// TIA Portal V18 export
FUNCTION_BLOCK "ST10_Flow14_B2Press"   // FB1084, GRAPH
// stored: AcknowledgeErrorsRequired false, AutoNumber false, GraphVersion 6.0, InitialValuesAcquisition false, SetENOAutomatically false
   // inherited from GRAPH_BASE
   VAR_INPUT
      iSysInface : "RCS_SysComInterface_V1";
   END_VAR
   VAR_IN_OUT
      ioPM_Inface : "RCS_PMInterface_V1";
      ioStatus : Int;
   END_VAR
   VAR
      sCtrlMode { S7_SetPoint := 'True'} : "SysFlowCtrlGraph";
      sUpdMES_Data : Bool;   // 更新MES数据
      工件放行中 : Bool;
      前站站号 { ExternalAccessible := 'False'; ExternalVisible := 'False'; ExternalWritable := 'False'} : UInt;
      本站站号 { ExternalAccessible := 'False'; ExternalVisible := 'False'; ExternalWritable := 'False'} : UInt;
      弹窗Temp : Array[1..10] of Int;
      AlarmID : Int;
      TON { S7_SetPoint := 'True'} : Array[0..10] of TON_TIME;
      TOF { S7_SetPoint := 'True'} : Array[0..10] of TOF_TIME;
      sUP { S7_SetPoint := 'True'} : Array[0..10] of Bool;
      更新RFID完成 : Bool;
   END_VAR
   VAR_TEMP
      Tempresult : USInt;
      本站站号乘10 : UInt;
   END_VAR
   // // TON[0] : 托盘流入1托盘到位传感器 / iA-Rotating product Check
   // // TON[1] : 托盘流入1托盘到位传感器
   // // TON[2] : 托盘流入1产品有无传感器
   // // TON[3] : 托盘流入1产品有无传感器
   // // TON[4] : 托盘流入1姿态检测光电2
   // // TON[5] : 托盘流入1姿态检测光电3
   // // TON[0].Q : 托盘流入1托盘到位 / iA-Rotating product Check
   // // TON[1].Q : 托盘流入1托盘无
   // // TON[2].Q : 托盘流入1有产品
   // // TON[3].Q : 托盘流入1无产品
   // // TON[4].Q : 托盘流入1姿态检测光电2
   // // TON[5].Q : 托盘流入1姿态检测光电3
   // // TOF[1] : iA-Rotating product Check
BEGIN
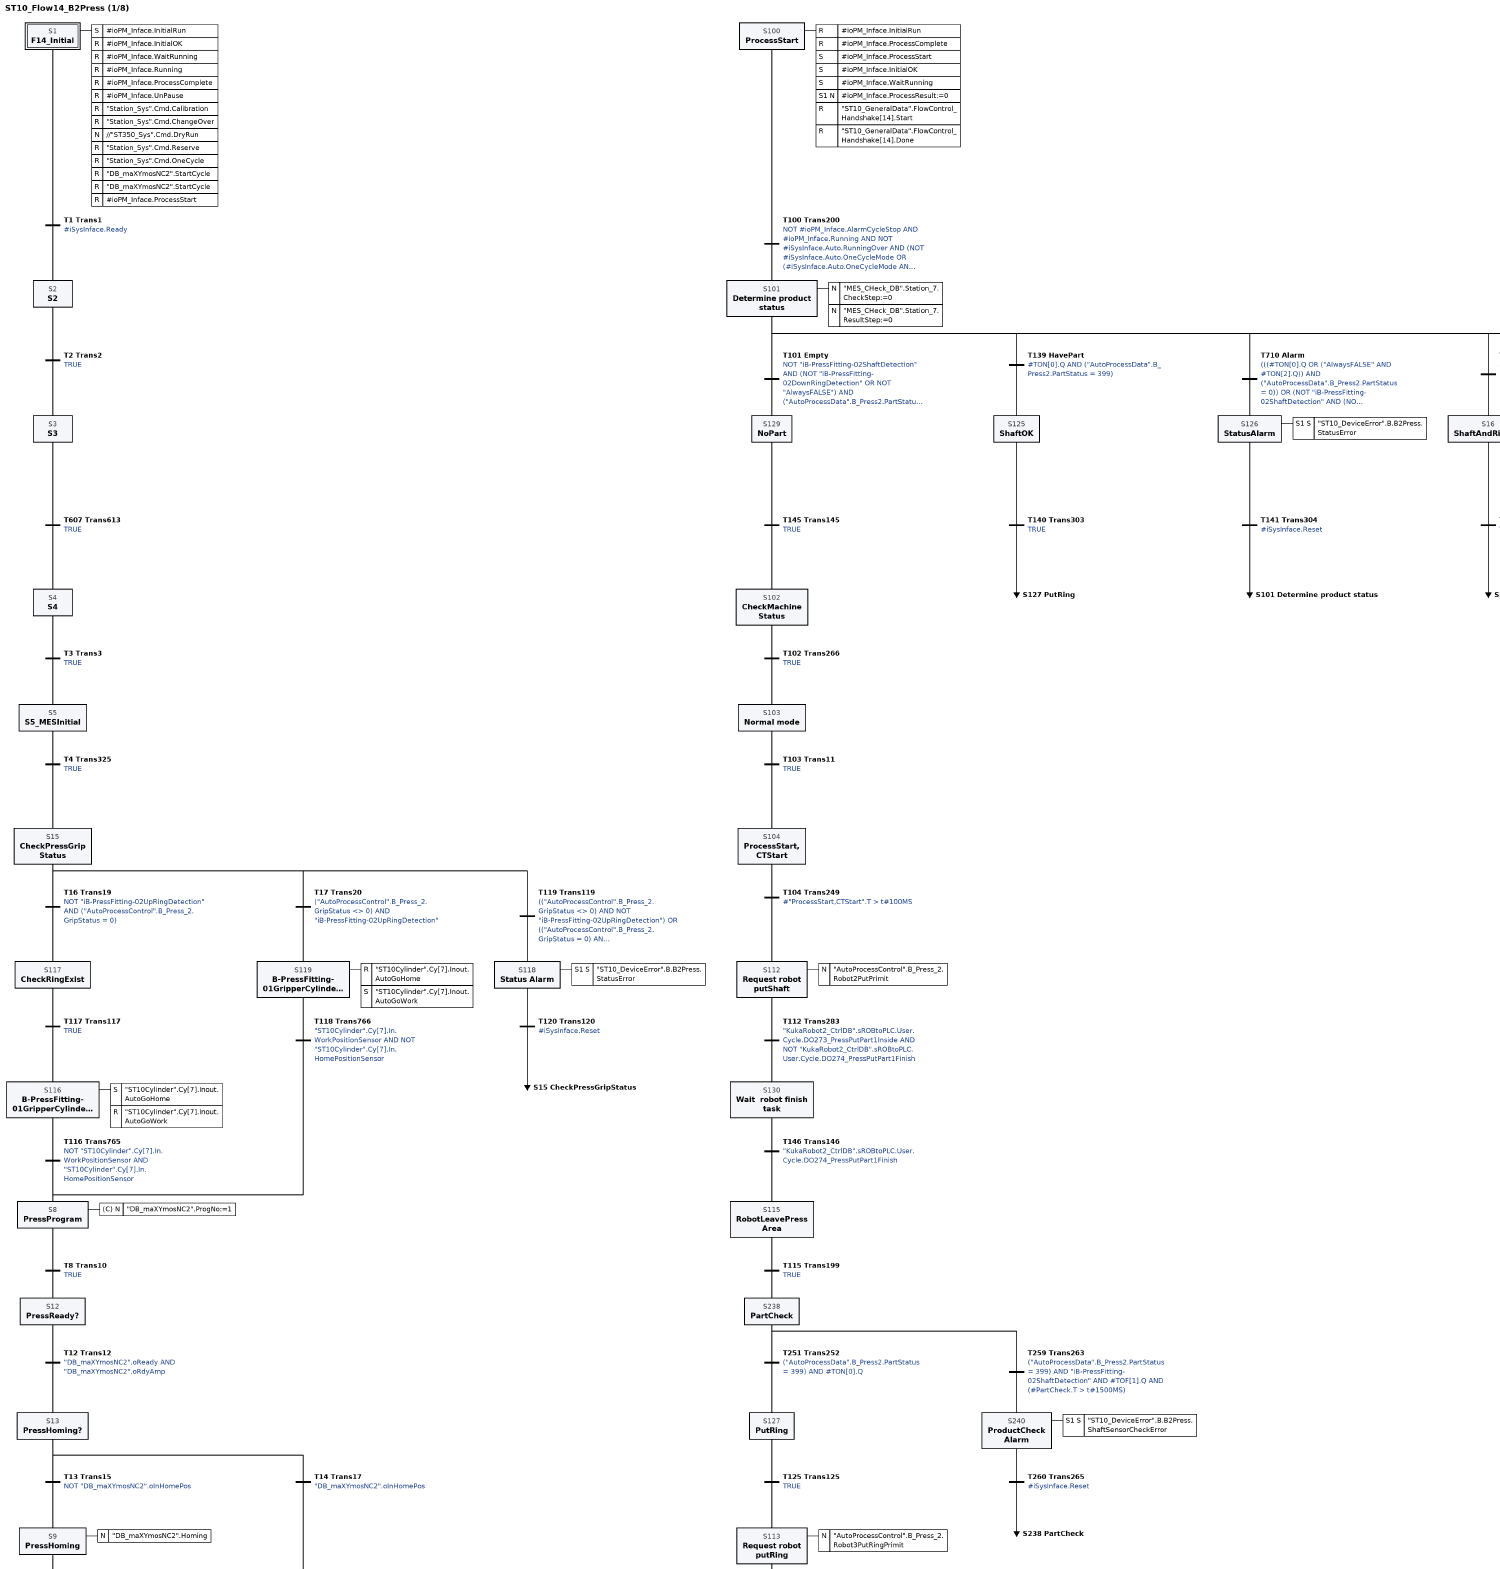
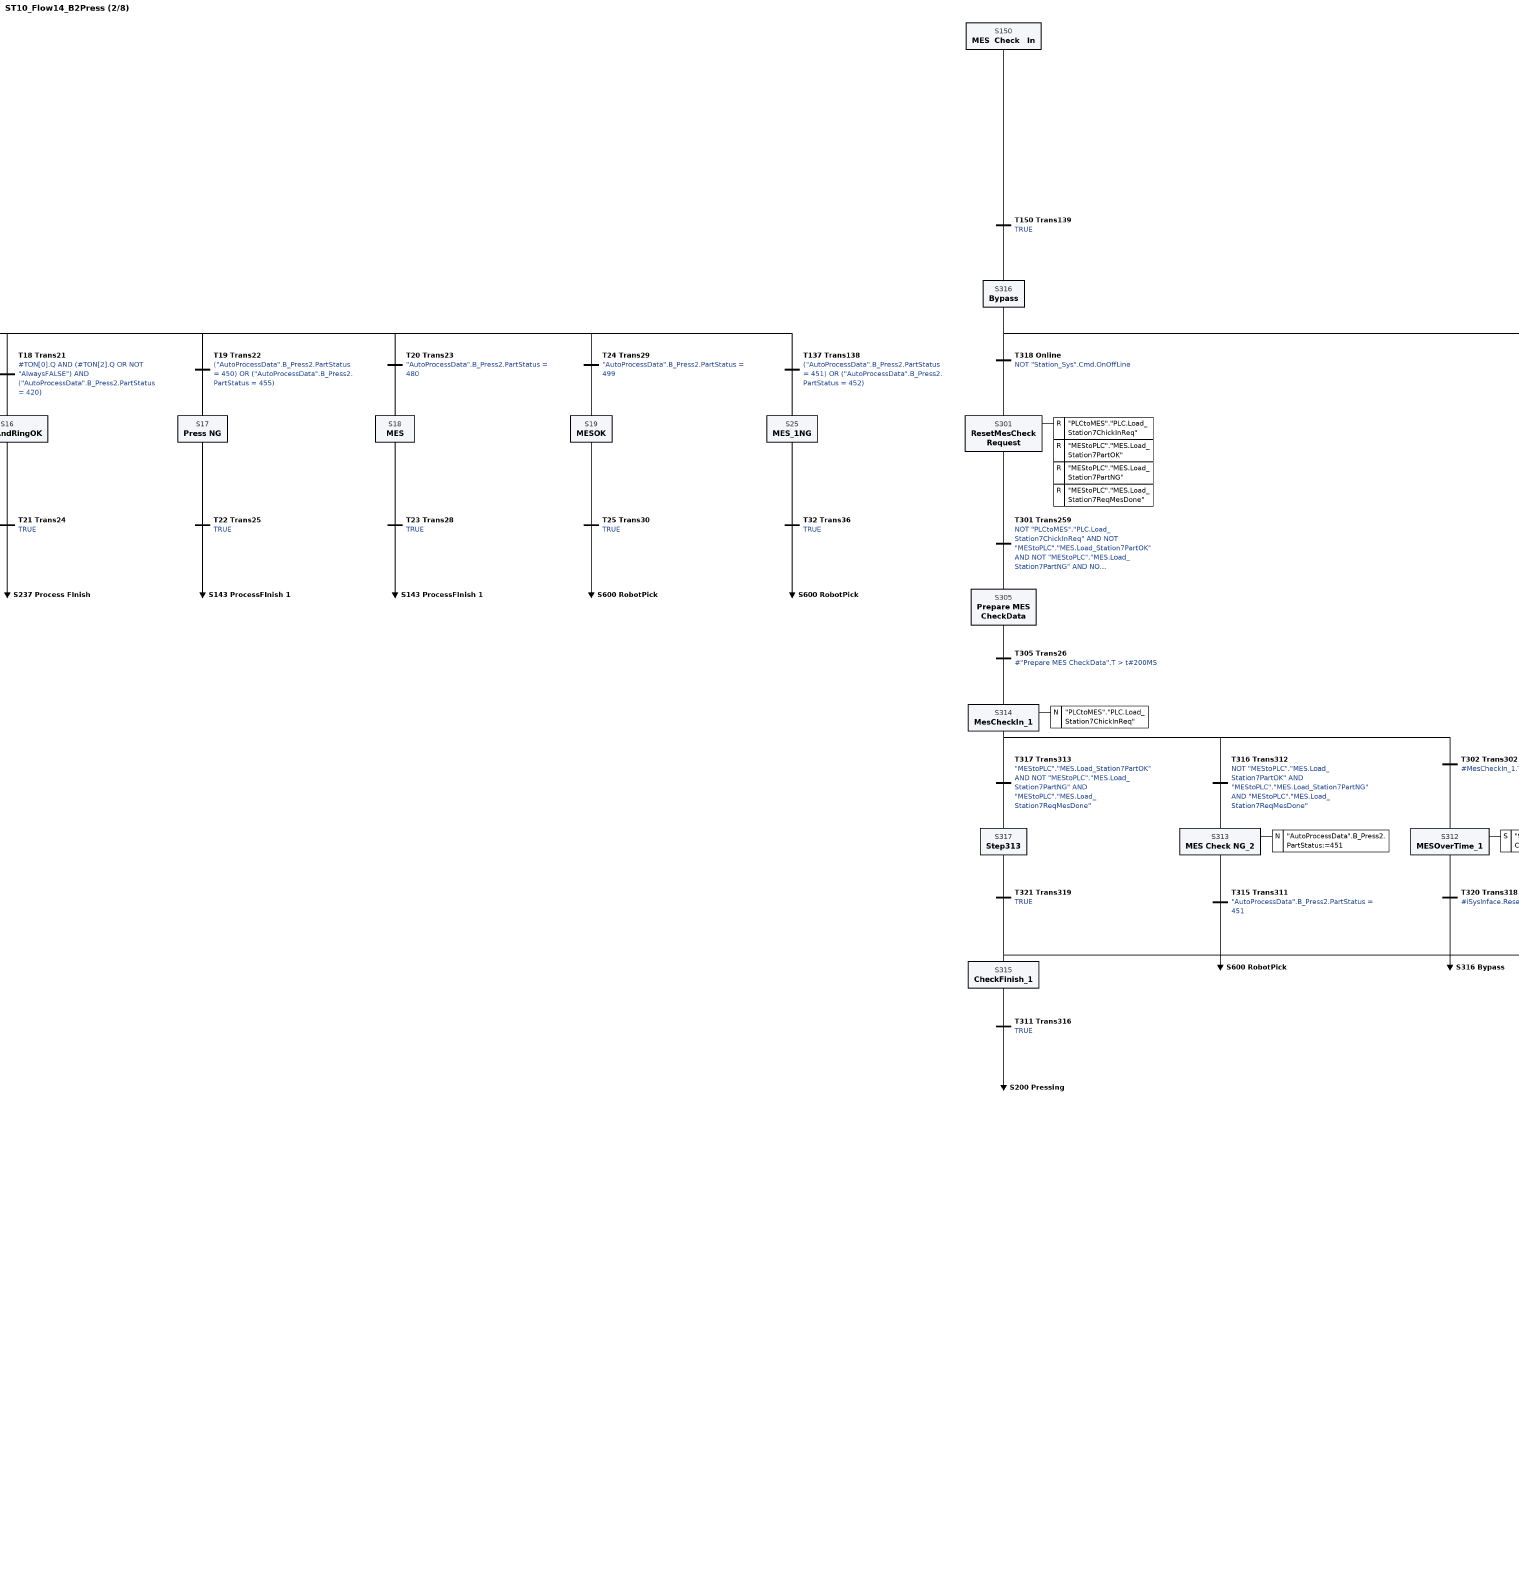
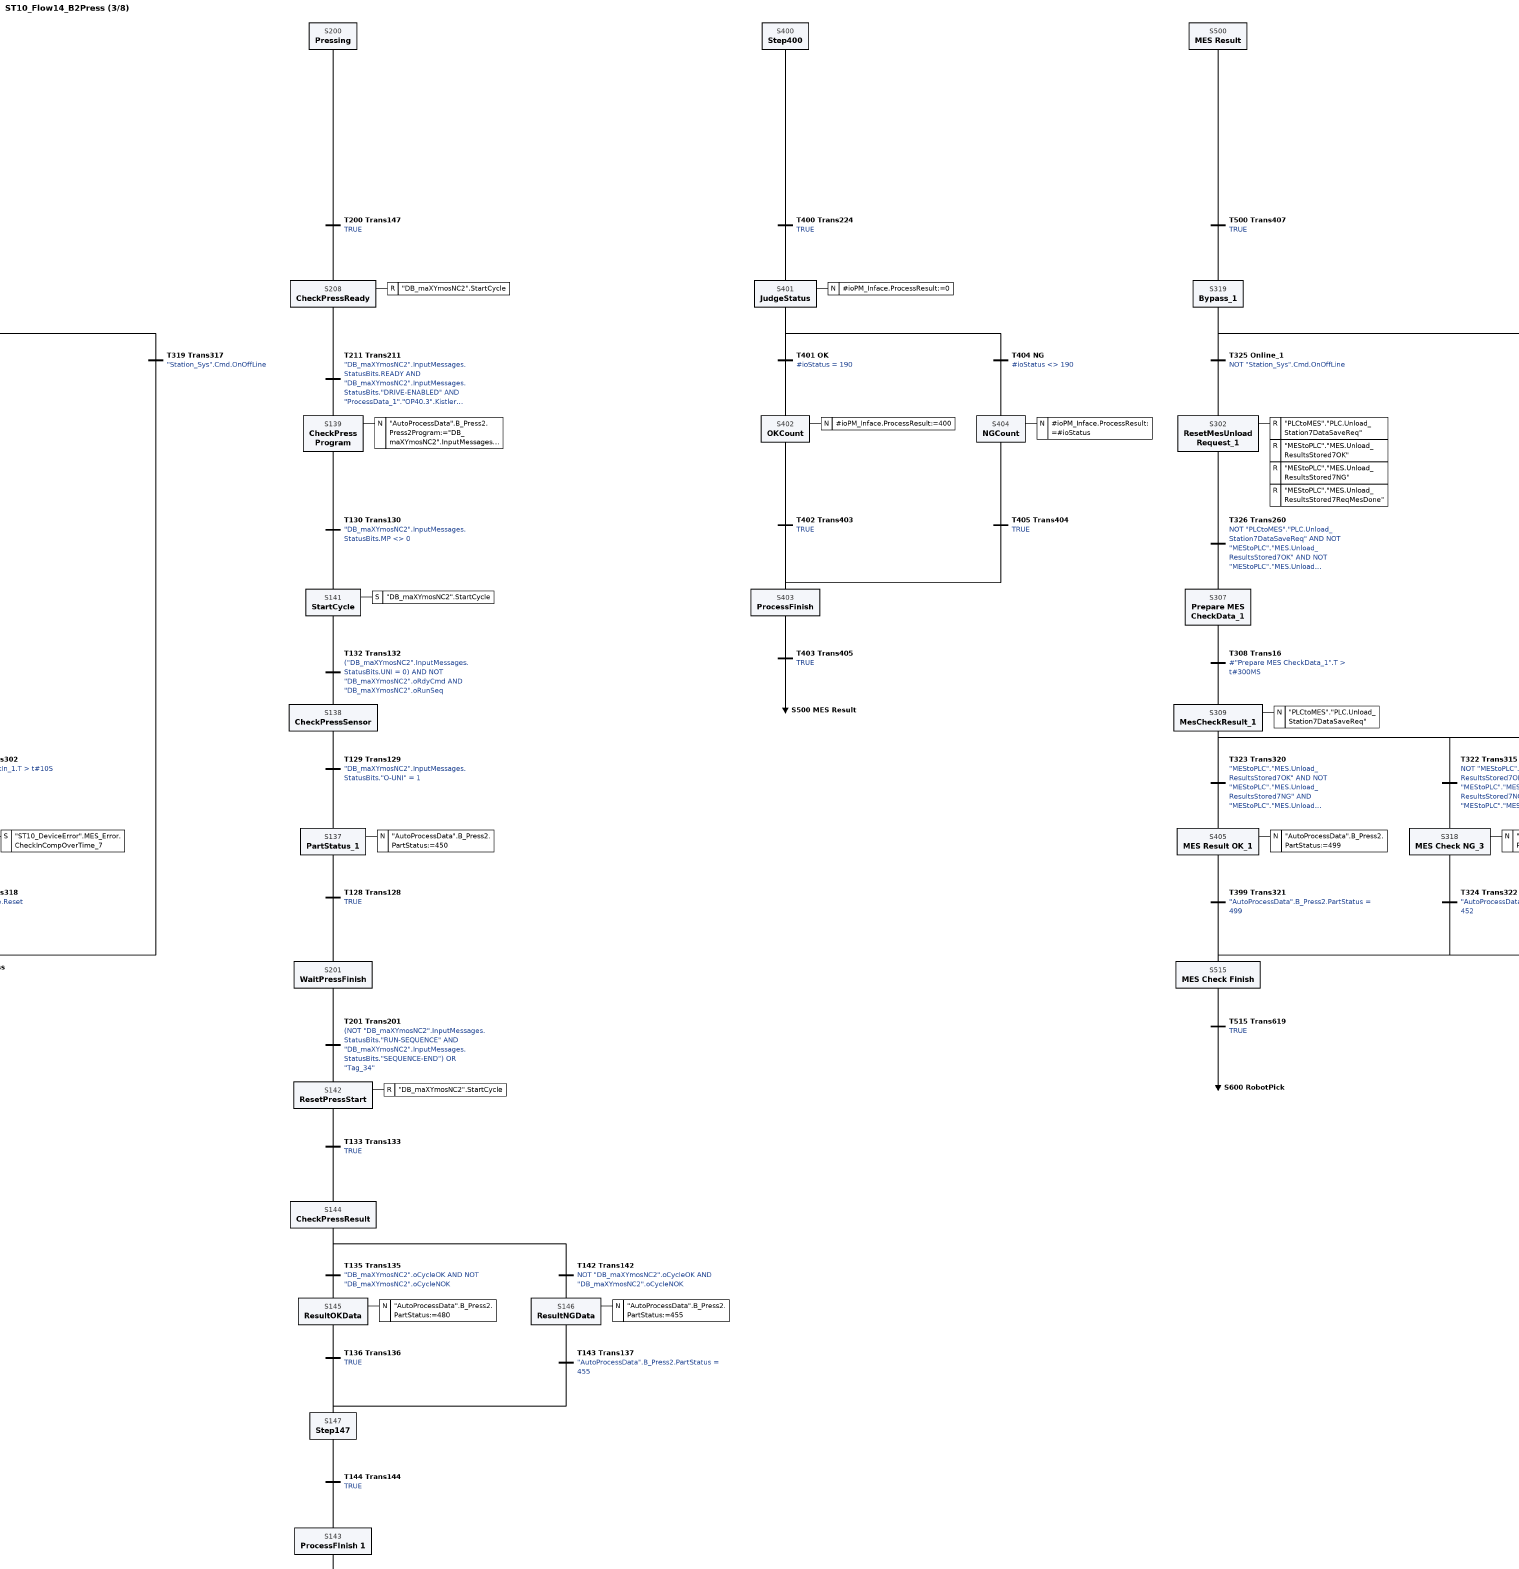
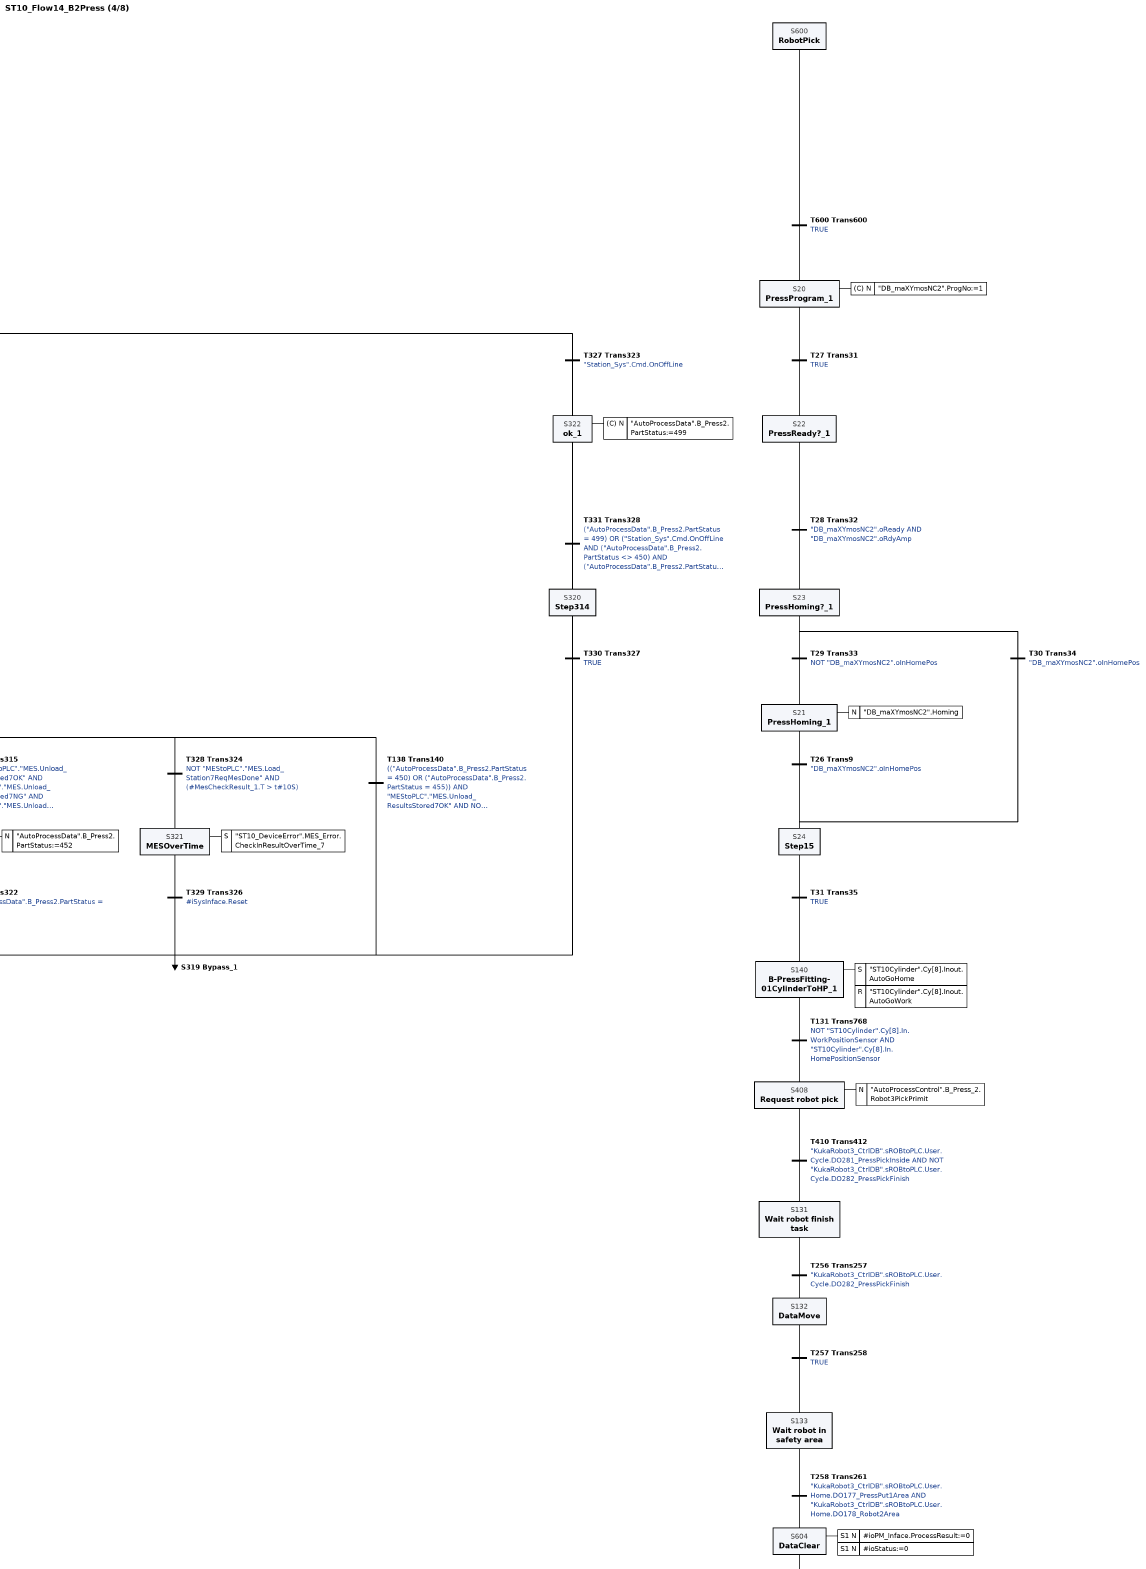
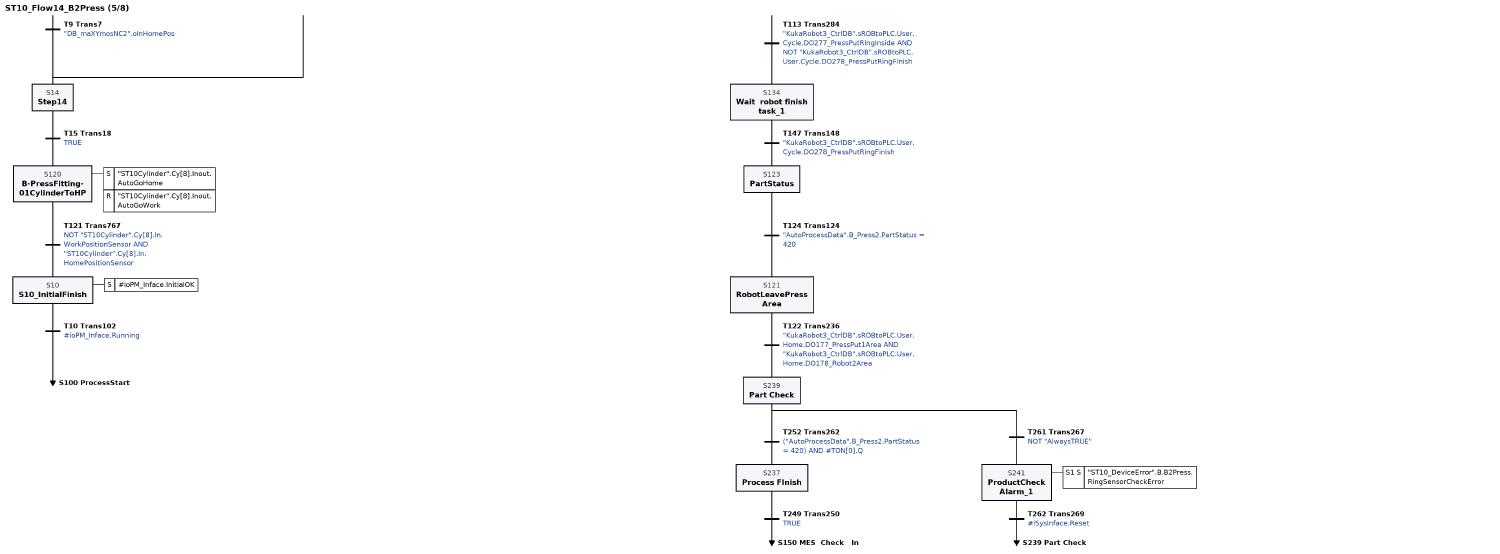
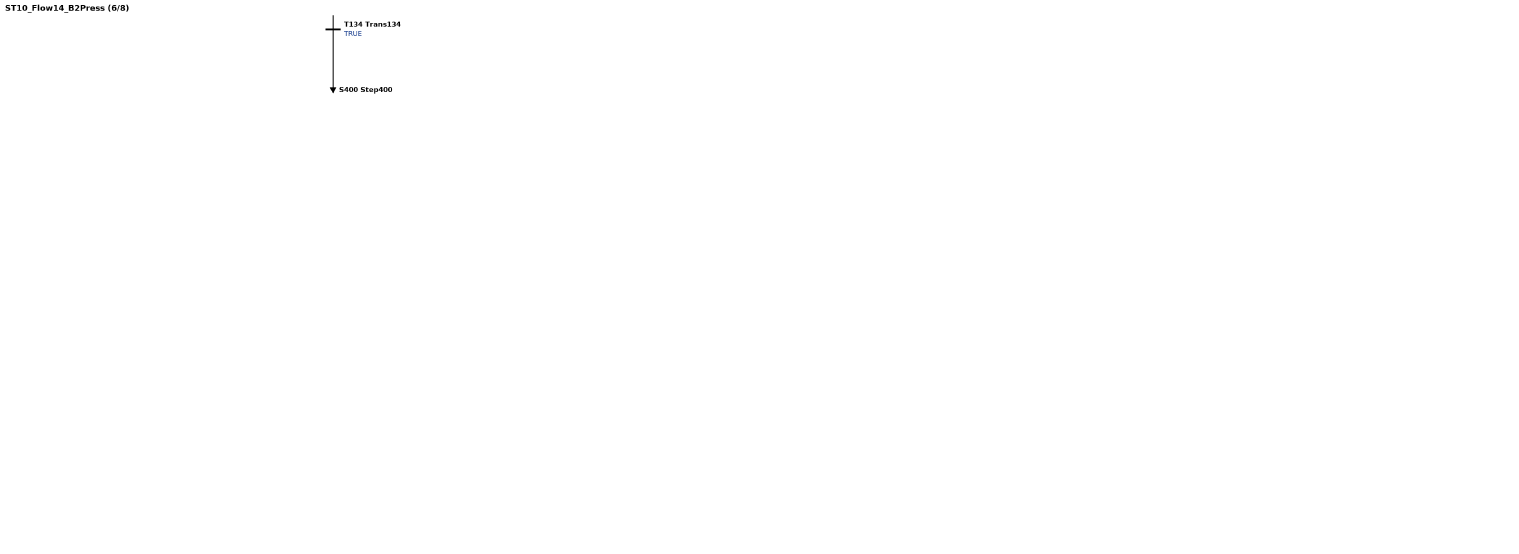
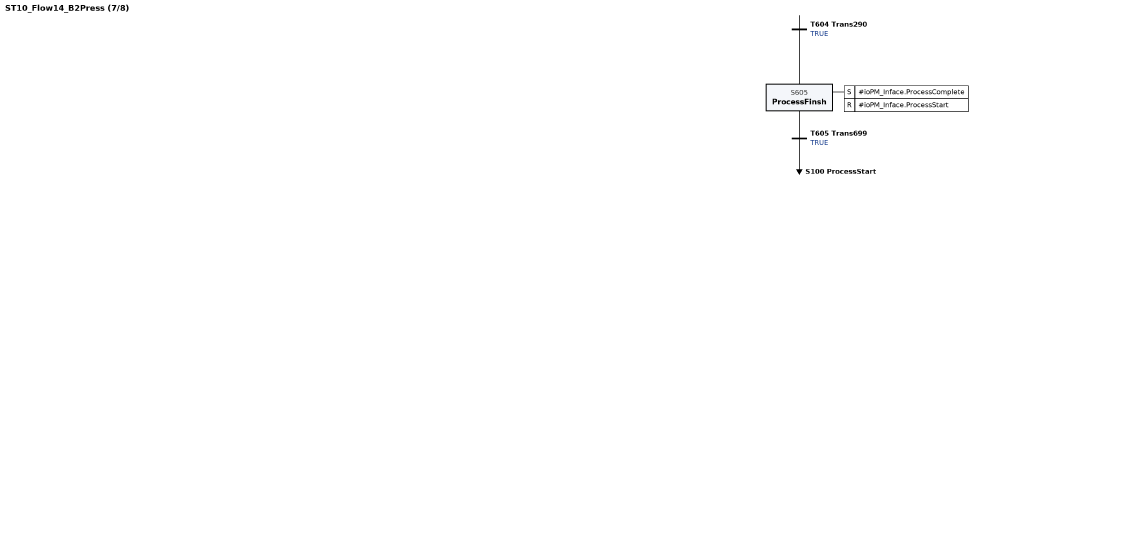
   // permanent pre-instructions
   NETWORK 1
      #TON[10].TON(IN := "AlwaysTRUE" AND "Station_Sys".Alarm.ImmediatelyStop, PT := T#300ms);
      #ioPM_Inface.AlarmImdilyStop := #TON[10].Q;
      #ioPM_Inface.AlarmCycleStop := "AlwaysTRUE" AND "Station_Sys".Alarm.CycleStop;
   NETWORK 2
      IF NOT False THEN
          #sCtrlMode(iSysInface := #iSysInface, ioPM_Inface := #ioPM_Inface, ioGraphCtrl := #RT_DATA.MOP);   // "SysFlowCtrlGraph"
      END_IF;
   NETWORK 3
      #TON[0].TON(IN := "AlwaysTRUE" AND "iB-PressFitting-02ShaftDetection", PT := t#500ms);   // 工位11有托盘
      #TOF[1].TOF(IN := "AlwaysTRUE" AND NOT "iB-PressFitting-02ShaftDetection", PT := T#300ms);   // 工位无托盘
      #TON[2].TON(IN := "AlwaysTRUE" AND "iB-PressFitting-02DownRingDetection", PT := T#300ms);
      #TOF[3].TOF(IN := "AlwaysTRUE" AND NOT "iB-PressFitting-02DownRingDetection", PT := T#300ms);
      #TON[4].TON(IN := "AlwaysTRUE" AND "iB-PressFitting-02UpRingDetection", PT := T#300ms);
      #TON[5].TON(IN := "AlwaysTRUE" AND NOT "iB-PressFitting-02UpRingDetection", PT := T#300ms);
   NETWORK 4
      #前站站号 := 345;
      #本站站号 := 350;

   // sequencer 1: S01-S99 初始化 / S01-S99 Initial
   INITIAL_STEP F14_Initial:   // S1, max time T#10S, warning time T#7S
              S    #ioPM_Inface.InitialRun
              R    #ioPM_Inface.InitialOK
              R    #ioPM_Inface.WaitRunning
              R    #ioPM_Inface.Running
              R    #ioPM_Inface.ProcessComplete
              R    #ioPM_Inface.UnPause
              R    "Station_Sys".Cmd.Calibration
              R    "Station_Sys".Cmd.ChangeOver
                   //"ST350_Sys".Cmd.DryRun
              R    "Station_Sys".Cmd.Reserve
              R    "Station_Sys".Cmd.OneCycle
              R    "DB_maXYmosNC2".StartCycle
              R    "DB_maXYmosNC2".StartCycle
              R    #ioPM_Inface.ProcessStart
              R    "AutoProcessControl".B_Press_2.Robot3PickPrimit
              R    "AutoProcessControl".B_Press_2.Robot3PutRingPrimit
              R    "AutoProcessControl".B_Press_2.Robot2PutPrimit
   END_STEP
   TRANSITION Trans1 FROM F14_Initial TO S2   // T1
      := #iSysInface.Ready;
   END_TRANSITION
   STEP S2:   // S2, max time T#10S, warning time T#7S
   END_STEP
   TRANSITION Trans2 FROM S2 TO S3   // T2
      := TRUE;
   END_TRANSITION
   STEP S4:   // S4, max time T#10S, warning time T#7S
   END_STEP
   TRANSITION Trans3 FROM S4 TO S5_MESInitial   // T3
      := TRUE;
   END_TRANSITION
   STEP S5_MESInitial:   // S5, max time T#10S, warning time T#7S
   END_STEP
   TRANSITION Trans325 FROM S5_MESInitial TO CheckPressGripStatus   // T4
      := TRUE;
   END_TRANSITION
   STEP S10_InitialFinish:   // S10, max time T#10S, warning time T#7S
              S    #ioPM_Inface.InitialOK
   END_STEP
   TRANSITION Trans102 FROM S10_InitialFinish TO ProcessStart   // T10, jump
      := #ioPM_Inface.Running;
   END_TRANSITION
   STEP S3:   // S3, max time T#10S, warning time T#7S
   END_STEP
   TRANSITION Trans613 FROM S3 TO S4   // T607
      := TRUE;
   END_TRANSITION
   STEP PressProgram:   // S8, max time T#10S, warning time T#7S
      interlock C := NOT "ST10_GeneralData".FunctionDeSelect."B".FunctionDeSelected_TestPress375A1;
      (C)     N    "DB_maXYmosNC2".ProgNo:=1
   END_STEP
   TRANSITION Trans10 FROM PressProgram TO "PressReady?"   // T8
      := TRUE;
   END_TRANSITION
   STEP PressHoming:   // S9, max time T#10S, warning time T#7S
              N    "DB_maXYmosNC2".Homing
   END_STEP
   TRANSITION Trans7 FROM PressHoming TO Step14   // T9
      := "DB_maXYmosNC2".oInHomePos;
   END_TRANSITION
   STEP "PressReady?":   // S12, max time T#10S, warning time T#7S
   END_STEP
   TRANSITION Trans12 FROM "PressReady?" TO "PressHoming?"   // T12
      := "DB_maXYmosNC2".oReady AND "DB_maXYmosNC2".oRdyAmp;
   END_TRANSITION
   STEP "PressHoming?":   // S13, max time T#10S, warning time T#7S
   END_STEP
   TRANSITION Trans15 FROM "PressHoming?" TO PressHoming   // T13
      := NOT "DB_maXYmosNC2".oInHomePos;
   END_TRANSITION
   TRANSITION Trans17 FROM "PressHoming?" TO Step14   // T14
      := "DB_maXYmosNC2".oInHomePos;
   END_TRANSITION
   STEP Step14:   // S14, max time T#10S, warning time T#7S
   END_STEP
   TRANSITION Trans18 FROM Step14 TO "B-PressFitting-01CylinderToHP"   // T15
      := TRUE;
   END_TRANSITION
   STEP CheckPressGripStatus:   // S15, max time T#10S, warning time T#7S
   END_STEP
   TRANSITION Trans19 FROM CheckPressGripStatus TO CheckRingExist   // T16
      := NOT "iB-PressFitting-02UpRingDetection" AND ("AutoProcessControl".B_Press_2.GripStatus = 0);
   END_TRANSITION
   TRANSITION Trans20 FROM CheckPressGripStatus TO "B-PressFitting-01GripperCylinderToWP"   // T17
      := ("AutoProcessControl".B_Press_2.GripStatus <> 0) AND "iB-PressFitting-02UpRingDetection";
   END_TRANSITION
   TRANSITION Trans119 FROM CheckPressGripStatus TO "Status Alarm"   // T119
      := (("AutoProcessControl".B_Press_2.GripStatus <> 0) AND NOT "iB-PressFitting-02UpRingDetection") OR (("AutoProcessControl".B_Press_2.GripStatus = 0) AND "iB-PressFitting-02UpRingDetection");
   END_TRANSITION
   STEP "B-PressFitting-01GripperCylinderToHP":   // S116, max time T#10S, warning time T#7S
              S    "ST10Cylinder".Cy[7].Inout.AutoGoHome
              R    "ST10Cylinder".Cy[7].Inout.AutoGoWork
   END_STEP
   TRANSITION Trans765 FROM "B-PressFitting-01GripperCylinderToHP" TO PressProgram   // T116
      := NOT "ST10Cylinder".Cy[7].In.WorkPositionSensor AND "ST10Cylinder".Cy[7].In.HomePositionSensor;
   END_TRANSITION
   STEP CheckRingExist:   // S117, max time T#10S, warning time T#7S
   END_STEP
   TRANSITION Trans117 FROM CheckRingExist TO "B-PressFitting-01GripperCylinderToHP"   // T117
      := TRUE;
   END_TRANSITION
   STEP "Status Alarm":   // S118, max time T#10S, warning time T#7S
          S1  S    "ST10_DeviceError".B.B2Press.StatusError
   END_STEP
   TRANSITION Trans120 FROM "Status Alarm" TO CheckPressGripStatus   // T120, jump
      := #iSysInface.Reset;
   END_TRANSITION
   STEP "B-PressFitting-01GripperCylinderToWP":   // S119, max time T#10S, warning time T#7S
              R    "ST10Cylinder".Cy[7].Inout.AutoGoHome
              S    "ST10Cylinder".Cy[7].Inout.AutoGoWork
   END_STEP
   TRANSITION Trans766 FROM "B-PressFitting-01GripperCylinderToWP" TO PressProgram   // T118
      := "ST10Cylinder".Cy[7].In.WorkPositionSensor AND NOT "ST10Cylinder".Cy[7].In.HomePositionSensor;
   END_TRANSITION
   STEP "B-PressFitting-01CylinderToHP":   // S120, max time T#10S, warning time T#7S
              S    "ST10Cylinder".Cy[8].Inout.AutoGoHome
              R    "ST10Cylinder".Cy[8].Inout.AutoGoWork
   END_STEP
   TRANSITION Trans767 FROM "B-PressFitting-01CylinderToHP" TO S10_InitialFinish   // T121
      := NOT "ST10Cylinder".Cy[8].In.WorkPositionSensor AND "ST10Cylinder".Cy[8].In.HomePositionSensor;
   END_TRANSITION

   // sequencer 2: S100-S199 等待到位 / S100-S149 CheckPartStatus
   STEP "Wait  robot finish task":   // S130, max time T#10S, warning time T#7S
   END_STEP
   TRANSITION Trans146 FROM "Wait  robot finish task" TO "RobotLeavePress Area"   // T146
      := "KukaRobot2_CtrlDB".sROBtoPLC.User.Cycle.DO274_PressPutPart1Finish;
   END_TRANSITION
   STEP CheckMachineStatus:   // S102, max time T#10S, warning time T#7S
   END_STEP
   TRANSITION Trans266 FROM CheckMachineStatus TO "Normal mode"   // T102
      := TRUE;
   END_TRANSITION
   STEP "Normal mode":   // S103, max time T#10S, warning time T#7S
   END_STEP
   TRANSITION Trans11 FROM "Normal mode" TO "ProcessStart,CTStart"   // T103
      := TRUE;
   END_TRANSITION
   STEP ProcessStart:   // S100, max time T#10S, warning time T#7S
      // 自动等待开始运行
              R    #ioPM_Inface.InitialRun
              R    #ioPM_Inface.ProcessComplete
              S    #ioPM_Inface.ProcessStart
              S    #ioPM_Inface.InitialOK
              S    #ioPM_Inface.WaitRunning
          S1  N    #ioPM_Inface.ProcessResult:=0
              R    "ST10_GeneralData".FlowControl_Handshake[14].Start
              R    "ST10_GeneralData".FlowControl_Handshake[14].Done
   END_STEP
   TRANSITION Trans200 FROM ProcessStart TO "Determine product status"   // T100
      := NOT #ioPM_Inface.AlarmCycleStop AND #ioPM_Inface.Running AND NOT #iSysInface.Auto.RunningOver AND (NOT #iSysInface.Auto.OneCycleMode OR (#iSysInface.Auto.OneCycleMode AND #ioPM_Inface.TriggerOneCycle));
   END_TRANSITION
   STEP "ProcessStart,CTStart":   // S104, max time T#10S, warning time T#7S
   END_STEP
   TRANSITION Trans249 FROM "ProcessStart,CTStart" TO "Request robot putShaft"   // T104
      := #"ProcessStart,CTStart".T > t#100MS;
   END_TRANSITION
   STEP "Process FInish":   // S237, max time T#10S, warning time T#7S
   END_STEP
   TRANSITION Trans250 FROM "Process FInish" TO "MES  Check   In"   // T249, jump
      := TRUE;
   END_TRANSITION
   STEP "Request robot putShaft":   // S112, max time T#10S, warning time T#7S
              N    "AutoProcessControl".B_Press_2.Robot2PutPrimit
   END_STEP
   TRANSITION Trans283 FROM "Request robot putShaft" TO "Wait  robot finish task"   // T112
      := "KukaRobot2_CtrlDB".sROBtoPLC.User.Cycle.DO273_PressPutPart1Inside AND NOT "KukaRobot2_CtrlDB".sROBtoPLC.User.Cycle.DO274_PressPutPart1Finish;
   END_TRANSITION
   STEP PutRing:   // S127, max time T#10S, warning time T#7S
   END_STEP
   TRANSITION Trans125 FROM PutRing TO "Request robot putRing"   // T125
      := TRUE;
   END_TRANSITION
   STEP PartCheck:   // S238, max time T#10S, warning time T#7S
   END_STEP
   TRANSITION Trans252 FROM PartCheck TO PutRing   // T251
      := ("AutoProcessData".B_Press2.PartStatus = 399) AND #TON[0].Q;
   END_TRANSITION
   TRANSITION Trans263 FROM PartCheck TO ProductCheckAlarm   // T259
      := ("AutoProcessData".B_Press2.PartStatus = 399) AND "iB-PressFitting-02ShaftDetection" AND #TOF[1].Q AND (#PartCheck.T > t#1500MS);
   END_TRANSITION
   STEP "Determine product status":   // S101, max time T#10S, warning time T#7S
              N    "MES_CHeck_DB".Station_7.CheckStep:=0
              N    "MES_CHeck_DB".Station_7.ResultStep:=0
   END_STEP
   TRANSITION Empty FROM "Determine product status" TO NoPart   // T101
      := NOT "iB-PressFitting-02ShaftDetection" AND (NOT "iB-PressFitting-02DownRingDetection" OR NOT "AlwaysFALSE") AND ("AutoProcessData".B_Press2.PartStatus = 0) AND (#"Determine product status".T > t#1000MS);
   END_TRANSITION
   TRANSITION HavePart FROM "Determine product status" TO ShaftOK   // T139
      := #TON[0].Q AND ("AutoProcessData".B_Press2.PartStatus = 399);
   END_TRANSITION
   TRANSITION Alarm FROM "Determine product status" TO StatusAlarm   // T710
      := (((#TON[0].Q OR ("AlwaysFALSE" AND #TON[2].Q)) AND ("AutoProcessData".B_Press2.PartStatus = 0)) OR (NOT "iB-PressFitting-02ShaftDetection" AND (NOT "iB-PressFitting-02DownRingDetection" OR NOT "AlwaysFALSE") AND ("AutoProcessData".B_Press2.PartStatus <> 0))) AND (#"Determine product status".T > t#1500MS);
   END_TRANSITION
   TRANSITION Trans21 FROM "Determine product status" TO ShaftAndRingOK   // T18
      := #TON[0].Q AND (#TON[2].Q OR NOT "AlwaysFALSE") AND ("AutoProcessData".B_Press2.PartStatus = 420);
   END_TRANSITION
   TRANSITION Trans22 FROM "Determine product status" TO "Press NG"   // T19
      := ("AutoProcessData".B_Press2.PartStatus = 450) OR ("AutoProcessData".B_Press2.PartStatus = 455);
   END_TRANSITION
   TRANSITION Trans23 FROM "Determine product status" TO MES   // T20
      := "AutoProcessData".B_Press2.PartStatus = 480;
   END_TRANSITION
   TRANSITION Trans29 FROM "Determine product status" TO MESOK   // T24
      := "AutoProcessData".B_Press2.PartStatus = 499;
   END_TRANSITION
   TRANSITION Trans138 FROM "Determine product status" TO MES_1NG   // T137
      := ("AutoProcessData".B_Press2.PartStatus = 451) OR ("AutoProcessData".B_Press2.PartStatus = 452);
   END_TRANSITION
   STEP ShaftOK:   // S125, max time T#10S, warning time T#7S
   END_STEP
   TRANSITION Trans303 FROM ShaftOK TO PutRing   // T140, jump
      := TRUE;
   END_TRANSITION
   STEP StatusAlarm:   // S126, max time T#10S, warning time T#7S
          S1  S    "ST10_DeviceError".B.B2Press.StatusError
   END_STEP
   TRANSITION Trans304 FROM StatusAlarm TO "Determine product status"   // T141, jump
      := #iSysInface.Reset;
   END_TRANSITION
   STEP NoPart:   // S129, max time T#10S, warning time T#7S
   END_STEP
   TRANSITION Trans145 FROM NoPart TO CheckMachineStatus   // T145
      := TRUE;
   END_TRANSITION
   STEP ShaftAndRingOK:   // S16, max time T#10S, warning time T#7S
   END_STEP
   TRANSITION Trans24 FROM ShaftAndRingOK TO "Process FInish"   // T21, jump
      := TRUE;
   END_TRANSITION
   STEP "Press NG":   // S17, max time T#10S, warning time T#7S
   END_STEP
   TRANSITION Trans25 FROM "Press NG" TO "ProcessFInish 1"   // T22, jump
      := TRUE;
   END_TRANSITION
   STEP MES:   // S18, max time T#10S, warning time T#7S
   END_STEP
   TRANSITION Trans28 FROM MES TO "ProcessFInish 1"   // T23, jump
      := TRUE;
   END_TRANSITION
   STEP MESOK:   // S19, max time T#10S, warning time T#7S
   END_STEP
   TRANSITION Trans30 FROM MESOK TO RobotPick   // T25, jump
      := TRUE;
   END_TRANSITION
   STEP "Wait  robot finish task_1":   // S134, max time T#10S, warning time T#7S
   END_STEP
   TRANSITION Trans148 FROM "Wait  robot finish task_1" TO PartStatus   // T147
      := "KukaRobot3_CtrlDB".sROBtoPLC.User.Cycle.DO278_PressPutRingFinish;
   END_TRANSITION
   STEP "Request robot putRing":   // S113, max time T#10S, warning time T#7S
              N    "AutoProcessControl".B_Press_2.Robot3PutRingPrimit
   END_STEP
   TRANSITION Trans284 FROM "Request robot putRing" TO "Wait  robot finish task_1"   // T113
      := "KukaRobot3_CtrlDB".sROBtoPLC.User.Cycle.DO277_PressPutRingInside AND NOT "KukaRobot3_CtrlDB".sROBtoPLC.User.Cycle.DO278_PressPutRingFinish;
   END_TRANSITION
   STEP "Part Check":   // S239, max time T#10S, warning time T#7S
   END_STEP
   TRANSITION Trans262 FROM "Part Check" TO "Process FInish"   // T252
      := ("AutoProcessData".B_Press2.PartStatus = 420) AND #TON[0].Q;
   END_TRANSITION
   TRANSITION Trans267 FROM "Part Check" TO ProductCheckAlarm_1   // T261
      := NOT "AlwaysTRUE";
   END_TRANSITION
   STEP ProductCheckAlarm:   // S240, max time T#10S, warning time T#7S
          S1  S    "ST10_DeviceError".B.B2Press.ShaftSensorCheckError
   END_STEP
   TRANSITION Trans265 FROM ProductCheckAlarm TO PartCheck   // T260, jump
      := #iSysInface.Reset;
   END_TRANSITION
   STEP ProductCheckAlarm_1:   // S241, max time T#10S, warning time T#7S
          S1  S    "ST10_DeviceError".B.B2Press.RingSensorCheckError
   END_STEP
   TRANSITION Trans269 FROM ProductCheckAlarm_1 TO "Part Check"   // T262, jump
      := #iSysInface.Reset;
   END_TRANSITION
   STEP RobotLeavePressArea:   // S121, max time T#10S, warning time T#7S
   END_STEP
   TRANSITION Trans236 FROM RobotLeavePressArea TO "Part Check"   // T122
      := "KukaRobot3_CtrlDB".sROBtoPLC.User.Home.DO177_PressPut1Area AND "KukaRobot3_CtrlDB".sROBtoPLC.User.Home.DO178_Robot2Area;
   END_TRANSITION
   STEP "RobotLeavePress Area":   // S115, max time T#10S, warning time T#7S
   END_STEP
   TRANSITION Trans199 FROM "RobotLeavePress Area" TO PartCheck   // T115
      := TRUE;
   END_TRANSITION
   STEP PartStatus:   // S123, max time T#10S, warning time T#7S
   END_STEP
   TRANSITION Trans124 FROM PartStatus TO RobotLeavePressArea   // T124
      := "AutoProcessData".B_Press2.PartStatus = 420;
   END_TRANSITION
   STEP MES_1NG:   // S25, max time T#10S, warning time T#7S
   END_STEP
   TRANSITION Trans36 FROM MES_1NG TO RobotPick   // T32, jump
      := TRUE;
   END_TRANSITION

   // sequencer 3: S150-S199 MES Check In
   STEP "MES  Check   In":   // S150, max time T#10S, warning time T#7S
   END_STEP
   TRANSITION Trans139 FROM "MES  Check   In" TO Bypass   // T150
      := TRUE;
   END_TRANSITION
   STEP MESOverTime_1:   // S312, max time T#10S, warning time T#7S
              S    "ST10_DeviceError".MES_Error.CheckInCompOverTime_7
   END_STEP
   TRANSITION Trans318 FROM MESOverTime_1 TO Bypass   // T320, jump
      := #iSysInface.Reset;
   END_TRANSITION
   STEP "MES Check NG_2":   // S313, max time T#10S, warning time T#7S
              N    "AutoProcessData".B_Press2.PartStatus:=451
   END_STEP
   TRANSITION Trans311 FROM "MES Check NG_2" TO RobotPick   // T315, jump
      := "AutoProcessData".B_Press2.PartStatus = 451;
   END_TRANSITION
   STEP ResetMesCheckRequest:   // S301, max time T#10S, warning time T#7S
              R    "PLCtoMES"."PLC.Load_Station7ChickInReq"
              R    "MEStoPLC"."MES.Load_Station7PartOK"
              R    "MEStoPLC"."MES.Load_Station7PartNG"
              R    "MEStoPLC"."MES.Load_Station7ReqMesDone"
   END_STEP
   TRANSITION Trans259 FROM ResetMesCheckRequest TO "Prepare MES CheckData"   // T301
      := NOT "PLCtoMES"."PLC.Load_Station7ChickInReq" AND NOT "MEStoPLC"."MES.Load_Station7PartOK" AND NOT "MEStoPLC"."MES.Load_Station7PartNG" AND NOT "MEStoPLC"."MES.Load_Station7ReqMesDone";
   END_TRANSITION
   STEP "Prepare MES CheckData":   // S305, max time T#10S, warning time T#7S
   END_STEP
   TRANSITION Trans26 FROM "Prepare MES CheckData" TO MesCheckIn_1   // T305
      := #"Prepare MES CheckData".T > t#200MS;
   END_TRANSITION
   STEP MesCheckIn_1:   // S314, max time T#10S, warning time T#7S
              N    "PLCtoMES"."PLC.Load_Station7ChickInReq"
   END_STEP
   TRANSITION Trans313 FROM MesCheckIn_1 TO Step313   // T317
      := "MEStoPLC"."MES.Load_Station7PartOK" AND NOT "MEStoPLC"."MES.Load_Station7PartNG" AND "MEStoPLC"."MES.Load_Station7ReqMesDone";
   END_TRANSITION
   TRANSITION Trans312 FROM MesCheckIn_1 TO "MES Check NG_2"   // T316
      := NOT "MEStoPLC"."MES.Load_Station7PartOK" AND "MEStoPLC"."MES.Load_Station7PartNG" AND "MEStoPLC"."MES.Load_Station7ReqMesDone";
   END_TRANSITION
   TRANSITION Trans302 FROM MesCheckIn_1 TO MESOverTime_1   // T302
      := #MesCheckIn_1.T > t#10S;
   END_TRANSITION
   STEP CheckFinish_1:   // S315, max time T#10S, warning time T#7S
   END_STEP
   TRANSITION Trans316 FROM CheckFinish_1 TO Pressing   // T311, jump
      := TRUE;
   END_TRANSITION
   STEP Bypass:   // S316, max time T#10S, warning time T#7S
   END_STEP
   TRANSITION Online FROM Bypass TO ResetMesCheckRequest   // T318
      := NOT "Station_Sys".Cmd.OnOffLine;
   END_TRANSITION
   TRANSITION Trans317 FROM Bypass TO CheckFinish_1   // T319
      := "Station_Sys".Cmd.OnOffLine;
   END_TRANSITION
   STEP Step313:   // S317, max time T#10S, warning time T#7S
   END_STEP
   TRANSITION Trans319 FROM Step313 TO CheckFinish_1   // T321
      := TRUE;
   END_TRANSITION

   // sequencer 4: S200-S299Pressing
   STEP Pressing:   // S200, max time T#10S, warning time T#7S
   END_STEP
   TRANSITION Trans147 FROM Pressing TO CheckPressReady   // T200
      := TRUE;
   END_TRANSITION
   STEP WaitPressFinish:   // S201, max time T#10S, warning time T#7S
   END_STEP
   TRANSITION Trans201 FROM WaitPressFinish TO ResetPressStart   // T201
      := (NOT "DB_maXYmosNC2".InputMessages.StatusBits."RUN-SEQUENCE" AND "DB_maXYmosNC2".InputMessages.StatusBits."SEQUENCE-END") OR "Tag_34";
   END_TRANSITION
   STEP ResultNGData:   // S146, max time T#10S, warning time T#7S
              N    "AutoProcessData".B_Press2.PartStatus:=455
   END_STEP
   TRANSITION Trans137 FROM ResultNGData TO Step147   // T143
      := "AutoProcessData".B_Press2.PartStatus = 455;
   END_TRANSITION
   STEP PartStatus_1:   // S137, max time T#10S, warning time T#7S
              N    "AutoProcessData".B_Press2.PartStatus:=450
   END_STEP
   TRANSITION Trans128 FROM PartStatus_1 TO WaitPressFinish   // T128
      := TRUE;
   END_TRANSITION
   STEP CheckPressSensor:   // S138, max time T#10S, warning time T#7S
   END_STEP
   TRANSITION Trans129 FROM CheckPressSensor TO PartStatus_1   // T129
      := "DB_maXYmosNC2".InputMessages.StatusBits."O-UNI" = 1;
   END_TRANSITION
   STEP ResetPressStart:   // S142, max time T#10S, warning time T#7S
              R    "DB_maXYmosNC2".StartCycle
   END_STEP
   TRANSITION Trans133 FROM ResetPressStart TO CheckPressResult   // T133
      := TRUE;
   END_TRANSITION
   STEP CheckPressProgram:   // S139, max time T#10S, warning time T#7S
              N    "AutoProcessData".B_Press2.Press2Program:="DB_maXYmosNC2".InputMessages.StatusBits.MP
   END_STEP
   TRANSITION Trans130 FROM CheckPressProgram TO StartCycle   // T130
      := "DB_maXYmosNC2".InputMessages.StatusBits.MP <> 0;
   END_TRANSITION
   STEP StartCycle:   // S141, max time T#10S, warning time T#7S
              S    "DB_maXYmosNC2".StartCycle
   END_STEP
   TRANSITION Trans132 FROM StartCycle TO CheckPressSensor   // T132
      := ("DB_maXYmosNC2".InputMessages.StatusBits.UNI = 0) AND NOT "DB_maXYmosNC2".oRdyCmd AND "DB_maXYmosNC2".oRunSeq;
   END_TRANSITION
   STEP CheckPressReady:   // S208, max time T#10S, warning time T#7S
              R    "DB_maXYmosNC2".StartCycle
   END_STEP
   TRANSITION Trans211 FROM CheckPressReady TO CheckPressProgram   // T211
      := "DB_maXYmosNC2".InputMessages.StatusBits.READY AND "DB_maXYmosNC2".InputMessages.StatusBits."DRIVE-ENABLED" AND "ProcessData_1"."OP40.3".Kistler_Interlock;
   END_TRANSITION
   STEP "ProcessFInish 1":   // S143, max time T#10S, warning time T#7S
   END_STEP
   TRANSITION Trans134 FROM "ProcessFInish 1" TO Step400   // T134, jump
      := TRUE;
   END_TRANSITION
   STEP ResultOKData:   // S145, max time T#10S, warning time T#7S
              N    "AutoProcessData".B_Press2.PartStatus:=480
   END_STEP
   TRANSITION Trans136 FROM ResultOKData TO Step147   // T136
      := TRUE;
   END_TRANSITION
   STEP CheckPressResult:   // S144, max time T#10S, warning time T#7S
   END_STEP
   TRANSITION Trans135 FROM CheckPressResult TO ResultOKData   // T135
      := "DB_maXYmosNC2".oCycleOK AND NOT "DB_maXYmosNC2".oCycleNOK;
   END_TRANSITION
   TRANSITION Trans142 FROM CheckPressResult TO ResultNGData   // T142
      := NOT "DB_maXYmosNC2".oCycleOK AND "DB_maXYmosNC2".oCycleNOK;
   END_TRANSITION
   STEP Step147:   // S147, max time T#10S, warning time T#7S
   END_STEP
   TRANSITION Trans144 FROM Step147 TO "ProcessFInish 1"   // T144
      := TRUE;
   END_TRANSITION

   // sequencer 5: S400-S499OK&NG数据处理 / S400-S499OK&NG Status Count
   STEP Step400:   // S400, max time T#10S, warning time T#7S
   END_STEP
   TRANSITION Trans224 FROM Step400 TO JudgeStatus   // T400
      := TRUE;
   END_TRANSITION
   STEP JudgeStatus:   // S401, max time T#10S, warning time T#7S
              N    #ioPM_Inface.ProcessResult:=0
   END_STEP
   TRANSITION OK FROM JudgeStatus TO OKCount   // T401
      := #ioStatus = 190;
   END_TRANSITION
   TRANSITION NG FROM JudgeStatus TO NGCount   // T404
      := #ioStatus <> 190;
   END_TRANSITION
   STEP OKCount:   // S402, max time T#10S, warning time T#7S
              N    #ioPM_Inface.ProcessResult:=400
   END_STEP
   TRANSITION Trans403 FROM OKCount TO ProcessFinish   // T402
      := TRUE;
   END_TRANSITION
   STEP NGCount:   // S404, max time T#10S, warning time T#7S
              N    #ioPM_Inface.ProcessResult:=#ioStatus
   END_STEP
   TRANSITION Trans404 FROM NGCount TO ProcessFinish   // T405
      := TRUE;
   END_TRANSITION
   STEP ProcessFinish:   // S403, max time T#10S, warning time T#7S
   END_STEP
   TRANSITION Trans405 FROM ProcessFinish TO "MES Result"   // T403, jump
      := TRUE;
   END_TRANSITION

   // sequencer 6: S500-S599 MES上传RFID写入 / S500-S599 MES Result
   STEP "MES Result":   // S500, max time T#10S, warning time T#7S
   END_STEP
   TRANSITION Trans407 FROM "MES Result" TO Bypass_1   // T500
      := TRUE;
   END_TRANSITION
   STEP "MES Check Finish":   // S515, max time T#10S, warning time T#7S
   END_STEP
   TRANSITION Trans619 FROM "MES Check Finish" TO RobotPick   // T515, jump
      := TRUE;
   END_TRANSITION
   STEP "MES Result OK_1":   // S405, max time T#10S, warning time T#7S
              N    "AutoProcessData".B_Press2.PartStatus:=499
   END_STEP
   TRANSITION Trans321 FROM "MES Result OK_1" TO "MES Check Finish"   // T399
      := "AutoProcessData".B_Press2.PartStatus = 499;
   END_TRANSITION
   STEP "MES Check NG_3":   // S318, max time T#10S, warning time T#7S
              N    "AutoProcessData".B_Press2.PartStatus:=452
   END_STEP
   TRANSITION Trans322 FROM "MES Check NG_3" TO "MES Check Finish"   // T324
      := "AutoProcessData".B_Press2.PartStatus = 452;
   END_TRANSITION
   STEP MesCheckResult_1:   // S309, max time T#10S, warning time T#7S
              N    "PLCtoMES"."PLC.Unload_Station7DataSaveReq"
   END_STEP
   TRANSITION Trans320 FROM MesCheckResult_1 TO "MES Result OK_1"   // T323
      := "MEStoPLC"."MES.Unload_ResultsStored7OK" AND NOT "MEStoPLC"."MES.Unload_ResultsStored7NG" AND "MEStoPLC"."MES.Unload_ResultsStored7ReqMesDone" AND ("AutoProcessData".B_Press2.PartStatus <> 450) AND ("AutoProcessData".B_Press2.PartStatus <> 455);
   END_TRANSITION
   TRANSITION Trans315 FROM MesCheckResult_1 TO "MES Check NG_3"   // T322
      := NOT "MEStoPLC"."MES.Unload_ResultsStored7OK" AND "MEStoPLC"."MES.Unload_ResultsStored7NG" AND "MEStoPLC"."MES.Unload_ResultsStored7ReqMesDone";
   END_TRANSITION
   TRANSITION Trans324 FROM MesCheckResult_1 TO MESOverTime   // T328
      := NOT "MEStoPLC"."MES.Load_Station7ReqMesDone" AND (#MesCheckResult_1.T > t#10S);
   END_TRANSITION
   TRANSITION Trans140 FROM MesCheckResult_1 TO "MES Check Finish"   // T138
      := (("AutoProcessData".B_Press2.PartStatus = 450) OR ("AutoProcessData".B_Press2.PartStatus = 455)) AND "MEStoPLC"."MES.Unload_ResultsStored7OK" AND NOT "MEStoPLC"."MES.Unload_ResultsStored7NG" AND "MEStoPLC"."MES.Unload_ResultsStored7ReqMesDone";
   END_TRANSITION
   STEP Bypass_1:   // S319, max time T#10S, warning time T#7S
   END_STEP
   TRANSITION Online_1 FROM Bypass_1 TO ResetMesUnloadRequest_1   // T325
      := NOT "Station_Sys".Cmd.OnOffLine;
   END_TRANSITION
   TRANSITION Trans323 FROM Bypass_1 TO ok_1   // T327
      := "Station_Sys".Cmd.OnOffLine;
   END_TRANSITION
   STEP ResetMesUnloadRequest_1:   // S302, max time T#10S, warning time T#7S
              R    "PLCtoMES"."PLC.Unload_Station7DataSaveReq"
              R    "MEStoPLC"."MES.Unload_ResultsStored7OK"
              R    "MEStoPLC"."MES.Unload_ResultsStored7NG"
              R    "MEStoPLC"."MES.Unload_ResultsStored7ReqMesDone"
   END_STEP
   TRANSITION Trans260 FROM ResetMesUnloadRequest_1 TO "Prepare MES CheckData_1"   // T326
      := NOT "PLCtoMES"."PLC.Unload_Station7DataSaveReq" AND NOT "MEStoPLC"."MES.Unload_ResultsStored7OK" AND NOT "MEStoPLC"."MES.Unload_ResultsStored7NG" AND NOT "MEStoPLC"."MES.Unload_ResultsStored7ReqMesDone";
   END_TRANSITION
   STEP Step314:   // S320, max time T#10S, warning time T#7S
   END_STEP
   TRANSITION Trans327 FROM Step314 TO "MES Check Finish"   // T330
      := TRUE;
   END_TRANSITION
   STEP MESOverTime:   // S321, max time T#10S, warning time T#7S
              S    "ST10_DeviceError".MES_Error.CheckInResultOverTime_7
   END_STEP
   TRANSITION Trans326 FROM MESOverTime TO Bypass_1   // T329, jump
      := #iSysInface.Reset;
   END_TRANSITION
   STEP ok_1:   // S322, max time T#10S, warning time T#7S
      interlock C := "AutoProcessData".B_Press2.PartStatus = 480;
      (C)     N    "AutoProcessData".B_Press2.PartStatus:=499
   END_STEP
   TRANSITION Trans328 FROM ok_1 TO Step314   // T331
      := ("AutoProcessData".B_Press2.PartStatus = 499) OR ("Station_Sys".Cmd.OnOffLine AND ("AutoProcessData".B_Press2.PartStatus <> 450) AND ("AutoProcessData".B_Press2.PartStatus <> 455));
   END_TRANSITION
   STEP "Prepare MES CheckData_1":   // S307, max time T#10S, warning time T#7S
   END_STEP
   TRANSITION Trans16 FROM "Prepare MES CheckData_1" TO MesCheckResult_1   // T308
      := #"Prepare MES CheckData_1".T > t#300MS;
   END_TRANSITION

   // sequencer 7: S600-S699工件放行 / S600-S699 RobotPick
   STEP RobotPick:   // S600, max time T#10S, warning time T#7S
   END_STEP
   TRANSITION Trans600 FROM RobotPick TO PressProgram_1   // T600
      := TRUE;
   END_TRANSITION
   STEP ProcessFinsh:   // S605, max time T#10S, warning time T#7S: 正式使用时，需要激活复位空循环
              S    #ioPM_Inface.ProcessComplete
              R    #ioPM_Inface.ProcessStart
   END_STEP
   TRANSITION Trans699 FROM ProcessFinsh TO ProcessStart   // T605, jump
      := TRUE;
   END_TRANSITION
   STEP DataClear:   // S604, max time T#10S, warning time T#7S
          S1  N    #ioPM_Inface.ProcessResult:=0
          S1  N    #ioStatus:=0
   END_STEP
   TRANSITION Trans290 FROM DataClear TO ProcessFinsh   // T604
      := TRUE;
   END_TRANSITION
   STEP "Request robot pick":   // S408, max time T#10S, warning time T#7S
              N    "AutoProcessControl".B_Press_2.Robot3PickPrimit
   END_STEP
   TRANSITION Trans412 FROM "Request robot pick" TO "Wait robot finish task"   // T410
      := "KukaRobot3_CtrlDB".sROBtoPLC.User.Cycle.DO281_PressPickInside AND NOT "KukaRobot3_CtrlDB".sROBtoPLC.User.Cycle.DO282_PressPickFinish;
   END_TRANSITION
   STEP "Wait robot finish task":   // S131, max time T#10S, warning time T#7S
   END_STEP
   TRANSITION Trans257 FROM "Wait robot finish task" TO DataMove   // T256
      := "KukaRobot3_CtrlDB".sROBtoPLC.User.Cycle.DO282_PressPickFinish;
   END_TRANSITION
   STEP DataMove:   // S132, max time T#10S, warning time T#7S
   END_STEP
   TRANSITION Trans258 FROM DataMove TO "Wait robot in safety area"   // T257
      := TRUE;
   END_TRANSITION
   STEP "Wait robot in safety area":   // S133, max time T#10S, warning time T#7S
   END_STEP
   TRANSITION Trans261 FROM "Wait robot in safety area" TO DataClear   // T258
      := "KukaRobot3_CtrlDB".sROBtoPLC.User.Home.DO177_PressPut1Area AND "KukaRobot3_CtrlDB".sROBtoPLC.User.Home.DO178_Robot2Area;
   END_TRANSITION
   STEP PressProgram_1:   // S20, max time T#10S, warning time T#7S
      interlock C := NOT "ST10_GeneralData".FunctionDeSelect."B".FunctionDeSelected_TestPress375A1;
      (C)     N    "DB_maXYmosNC2".ProgNo:=1
   END_STEP
   TRANSITION Trans31 FROM PressProgram_1 TO "PressReady?_1"   // T27
      := TRUE;
   END_TRANSITION
   STEP PressHoming_1:   // S21, max time T#10S, warning time T#7S
              N    "DB_maXYmosNC2".Homing
   END_STEP
   TRANSITION Trans9 FROM PressHoming_1 TO Step15   // T26
      := "DB_maXYmosNC2".oInHomePos;
   END_TRANSITION
   STEP "PressReady?_1":   // S22, max time T#10S, warning time T#7S
   END_STEP
   TRANSITION Trans32 FROM "PressReady?_1" TO "PressHoming?_1"   // T28
      := "DB_maXYmosNC2".oReady AND "DB_maXYmosNC2".oRdyAmp;
   END_TRANSITION
   STEP "PressHoming?_1":   // S23, max time T#10S, warning time T#7S
   END_STEP
   TRANSITION Trans33 FROM "PressHoming?_1" TO PressHoming_1   // T29
      := NOT "DB_maXYmosNC2".oInHomePos;
   END_TRANSITION
   TRANSITION Trans34 FROM "PressHoming?_1" TO Step15   // T30
      := "DB_maXYmosNC2".oInHomePos;
   END_TRANSITION
   STEP Step15:   // S24, max time T#10S, warning time T#7S
   END_STEP
   TRANSITION Trans35 FROM Step15 TO "B-PressFitting-01CylinderToHP_1"   // T31
      := TRUE;
   END_TRANSITION
   STEP "B-PressFitting-01CylinderToHP_1":   // S140, max time T#10S, warning time T#7S
              S    "ST10Cylinder".Cy[8].Inout.AutoGoHome
              R    "ST10Cylinder".Cy[8].Inout.AutoGoWork
   END_STEP
   TRANSITION Trans768 FROM "B-PressFitting-01CylinderToHP_1" TO "Request robot pick"   // T131
      := NOT "ST10Cylinder".Cy[8].In.WorkPositionSensor AND "ST10Cylinder".Cy[8].In.HomePositionSensor;
   END_TRANSITION

   // permanent post-instructions
   NETWORK 1
      #ioPM_Inface.StepNum := #RT_DATA.S_DISPLAY;
   NETWORK 2
      IF #iSysInface.Reset THEN #AlarmID := 0; END_IF;
   NETWORK 3
      #TON[10].TON(IN := #工件放行中, PT := T#0.5S);
      IF #TON[10].Q THEN #工件放行中 := FALSE; END_IF;
END_FUNCTION_BLOCK
